// TIA Portal V19 export
// export: Created 2026-08-08T14:07:57.97432Z, ExportSetting WithDefaults, DisplayName Totally Integrated Automation Portal, DisplayVersion V19, DisplayName TIA Portal Openness, DisplayVersion V19, DisplayName TIA Portal Version Control Interface, DisplayVersion V19, DisplayName STEP 7 Professional, DisplayVersion V19, DisplayName STEP 7 Safety, DisplayVersion V19, DisplayName WinCC Basic/Comfort/Advanced, DisplayVersion V19, DisplayName WinCC Unified, DisplayVersion V19
DATA_BLOCK "ceD"   // DB1
{ S7_Optimized_Access := 'TRUE' }
VERSION : 0.1
// stored: AutoNumber true, DBAccessibleFromOPCUA true, DBAccessibleFromWebserver true, IsOnlyStoredInLoadMemory false, IsRetainMemResEnabled false, IsWriteProtectedInAS false, MemoryReserve 100
   VAR
      IN : Struct
         in1 : Bool;
         in2 : Int;
         in3 : Int;
         in4 : Int;
         in5 : Bool;
      END_STRUCT;
      out : Struct
         out1 : Bool;
         out2 : Int;
         out3 : Int;
      END_STRUCT;
   END_VAR
BEGIN
END_DATA_BLOCK
